FUNCTION_BLOCK CROSSCOMM_PEER_7809690FA4BAE57E (* Service Interface Function Block Type *)
  (* Standard: 61499-2 *)
  (* Version 0.0, 9/22/2017, bababen, nxtControl GmbH, template *)
  PACKAGE Main;
  (* Compiler Cpp nxtControl builtin 1.0 *)
  {SET_ATTRIBUTE(Runtime.FBType.ImplementingType, Runtime.System#DYNGEN_CROSSCOMM_PEER)}
  {SET_ATTRIBUTE(Configuration.GenericFBType.InterfaceParams, Runtime.System#<InterfaceList> <EventOutputs> <Event Name="IND"> <With Var="VAL" /> </Event> </EventOutputs> <OutputVars> <VarDeclaration Name="VAL" Type="BOOL" /> </OutputVars> </InterfaceList>)}
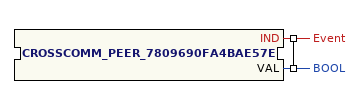
  EVENT_OUTPUT
    IND WITH VAL;
  END_EVENT
  VAR_OUTPUT
    VAL : BOOL;
  END_VAR
  EC_STATES
    START;
  END_STATES
END_FUNCTION_BLOCK
